Fanuc KAREL source: port_TPOUT.kl

PROGRAM TP
%NOLOCKGROUP
VAR
 x: BOOLEAN
BEGIN
 x = TPOUT[3]
END TP
